// TwinCAT 3 PLC project SortingConveyor
// ProgramVersion: 3.1.4024.0
// libraries:
//   Tc2_Standard, * (Beckhoff Automation GmbH)
//   Tc2_System, * (Beckhoff Automation GmbH)
//   Tc3_Module, * (Beckhoff Automation GmbH)
// project tree:
//   / PlcTask.TcTTO
//   POUs/ MAIN.TcPOU

CONFIGURATION SortingConveyor
    RESOURCE PLC ON TwinCAT3
        TASK PlcTask(INTERVAL := T#10ms, PRIORITY := 24);
        PROGRAM MAIN WITH PlcTask : MAIN;
    END_RESOURCE
END_CONFIGURATION

// ---- POUs/MAIN.TcPOU
PROGRAM MAIN
VAR
	bBadPartDetected: BOOL := FALSE;
	bRejectArmEnabled: BOOL := FALSE;
	tTravelTimer: TON;
	tPushTimer: TON;
	bRejectMemory: BOOL := FALSE;
	
END_VAR

IF bBadPartDetected THEN
	bRejectMemory := TRUE;
END_IF;
tTravelTimer(IN:= bRejectMemory, PT := T#3S);
tPushTimer(IN:= tTravelTimer.Q, PT:= T#1S);
IF NOT tPushTimer.Q AND bRejectMemory AND tTravelTimer.Q THEN
	bRejectArmEnabled := TRUE;
ELSE;
	bRejectArmEnabled := FALSE;
END_IF;
IF tPushTimer.Q AND tTravelTimer.Q THEN
	bBadPartDetected := FALSE;
	bRejectMemory := FALSE;
END_IF;

END_PROGRAM
